Yaskawa INFORM job: 25P.JBI

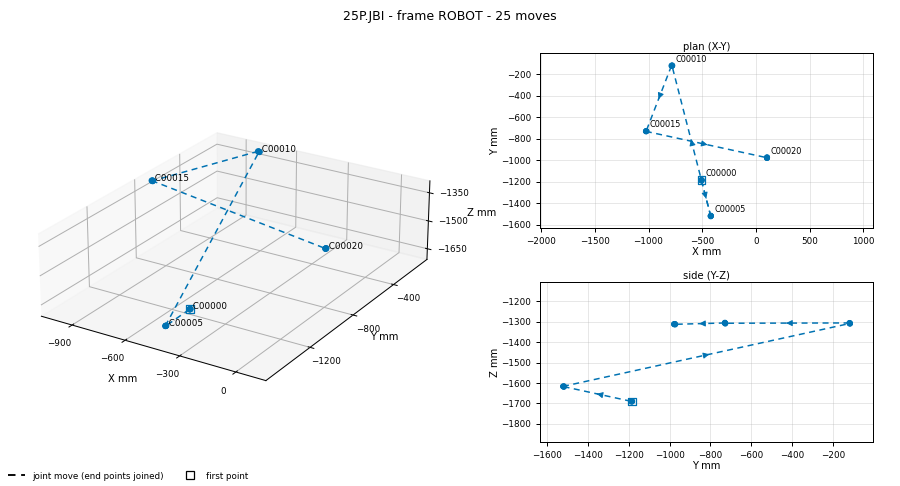
[picture p0: tool path of 25P.JBI in frame ROBOT, 25 of 25 moves have a stored position in this frame; points joined in program order, loops and branches not executed]
/JOB
//NAME 25P
///FOLDERNAME INNE
//POS
///NPOS 25,25,0,0,0,0
///TOOL 0
///POSTYPE ROBOT
///RECTAN
///RCONF 0,0,0,0,0,0,0,0,0,0,0,0,0,0,0,0,0,0,0,0,0,0,0,0
C00000=-507.342,-1184.581,-1690.032,-0.0187,0.0172,165.3916
C00001=-506.975,-1184.439,-1690.036,27.4910,6.8900,167.0984
C00002=-506.471,-1184.506,-1689.976,-21.9037,-5.5324,166.4486
C00003=-505.654,-1182.490,-1689.130,-10.3952,34.6465,162.1420
C00004=-507.341,-1188.850,-1689.091,10.5220,-35.0774,162.0592
C00005=-420.627,-1517.311,-1617.530,-0.0014,0.0208,165.3779
C00006=-420.913,-1517.651,-1616.420,31.0796,7.6818,167.5378
C00007=-420.839,-1517.434,-1617.483,-12.8806,-3.3043,165.7525
C00008=-419.594,-1515.066,-1616.962,-9.7805,33.0538,162.4549
C00009=-420.792,-1521.243,-1616.425,9.5715,-32.5378,162.5857
C00010=-782.092,-117.419,-1308.421,-0.0034,-0.0013,121.9949
C00011=-778.858,-117.694,-1309.179,13.3188,20.2463,124.3838
C00012=-782.680,-118.524,-1308.667,-15.4039,-23.0332,125.1487
C00013=-779.592,-119.939,-1306.947,-25.2512,14.9184,118.6361
C00014=-786.551,-119.756,-1306.067,24.8946,-14.7401,118.7234
C00015=-1021.944,-727.921,-1307.561,-0.0041,-0.0003,150.7974
C00016=-1020.832,-727.415,-1309.296,32.4761,16.7095,155.6935
C00017=-1020.818,-728.614,-1307.106,-25.7957,-13.6711,153.9361
C00018=-1020.072,-729.138,-1304.844,-18.7418,29.8844,145.7553
C00019=-1024.761,-730.018,-1306.239,17.1823,-27.8610,146.5071
C00020=101.665,-975.279,-1312.797,-0.0009,-0.0013,-141.4418
C00021=102.596,-978.667,-1312.063,22.3464,-16.8630,-144.7952
C00022=103.966,-973.729,-1310.810,-21.2601,16.1189,-144.4830
C00023=103.033,-972.056,-1313.466,25.1611,28.0860,-135.0569
C00024=102.493,-976.093,-1312.305,-22.4305,-25.5818,-136.2952
BC00000=1343.240,419.551,636.110
BC00001=1343.240,419.551,636.110
BC00002=1343.240,419.551,636.110
BC00003=1343.240,419.551,636.110
BC00004=1343.240,419.551,636.110
BC00005=1343.240,419.551,636.110
BC00006=1343.240,419.551,636.110
BC00007=1343.240,419.551,636.110
BC00008=1343.240,419.551,636.110
BC00009=1343.240,419.551,636.110
BC00010=1343.240,419.551,636.105
BC00011=1343.240,419.551,636.105
BC00012=1343.240,419.551,636.105
BC00013=1343.240,419.551,636.105
BC00014=1343.240,419.551,636.105
BC00015=1343.240,419.551,636.105
BC00016=1343.240,419.551,636.105
BC00017=1343.240,419.551,636.105
BC00018=1343.240,419.551,636.105
BC00019=1343.240,419.551,636.105
BC00020=1343.240,419.551,636.105
BC00021=1343.240,419.551,636.105
BC00022=1343.240,419.551,636.105
BC00023=1343.240,419.551,636.105
BC00024=1343.240,419.551,636.105
//INST
///DATE 2023/10/04 15:13
///ATTR SC,RW,RJ
////FRAME ROBOT
///GROUP1 RB1,BS1
NOP
MOVJ C00000 BC00000 VJ=0.78
MOVJ C00001 BC00001 VJ=0.78
MOVJ C00002 BC00002 VJ=0.78
MOVJ C00003 BC00003 VJ=0.78
MOVJ C00004 BC00004 VJ=0.78
MOVJ C00005 BC00005 VJ=0.78
MOVJ C00006 BC00006 VJ=0.78
MOVJ C00007 BC00007 VJ=0.78
MOVJ C00008 BC00008 VJ=0.78
MOVJ C00009 BC00009 VJ=0.78
MOVJ C00010 BC00010 VJ=0.78
MOVJ C00011 BC00011 VJ=0.78
MOVJ C00012 BC00012 VJ=0.78
MOVJ C00013 BC00013 VJ=0.78
MOVJ C00014 BC00014 VJ=0.78
MOVJ C00015 BC00015 VJ=0.78
MOVJ C00016 BC00016 VJ=0.78
MOVJ C00017 BC00017 VJ=0.78
MOVJ C00018 BC00018 VJ=0.78
MOVJ C00019 BC00019 VJ=0.78
MOVJ C00020 BC00020 VJ=0.78
MOVJ C00021 BC00021 VJ=0.78
MOVJ C00022 BC00022 VJ=0.78
MOVJ C00023 BC00023 VJ=0.78
MOVJ C00024 BC00024 VJ=0.78
END
